# EPICS autosave request: support/ebrick/2-2-3/iocBoot/iocebrick/autosave/ebrickSEN.req
$(P)$(H)$(F)$(D):dis
$(P)$(H)$(F)$(D):type
$(P)$(H)$(F)$(D):code
$(P)$(H)$(F)$(D):volt
$(P)$(H)$(F)$(D):resist
$(P)$(H)$(F)$(D):thermo
$(P)$(H)$(F)$(D):rtd
$(P)$(H)$(F)$(D):thermis
$(P)$(H)$(F)$(D):curr
#
$(P)$(H)$(F)$(D).SCAN
$(P)$(H)$(F)$(D).DESC
$(P)$(H)$(F)$(D).PREC
$(P)$(H)$(F)$(D).LOPR
$(P)$(H)$(F)$(D).HOPR
$(P)$(H)$(F)$(D).EGU
